PROGRAM ServoTronix
VAR_INPUT
	bExecute : REFERENCE TO BOOL;
END_VAR
VAR
	servo : AXIS_REF;
	
	mcPower : MC_Power;
	mcMoveVelocity : MC_MoveVelocity;
	mcSetPosition : MC_SetPosition;
	mcStop : MC_Stop;
	
	mcReset : MC_Reset;
	preset : BOOL;
	
	bReset : BOOL;
	positionSet : BOOL;
	
	randomPos : INT;
	
	homeLimit AT %I* : BOOL;
	home AT %I* : BOOL;
	travelLimit AT %I* : BOOL;
	
	step : (IDLE, HOME_BACK, HOME_FINAL, STOP, SET, FORWARD, REDO_HOME);
END_VAR

(*
IF NOT preset THEN
	preset := TRUE;
	bReset := TRUE;
END_IF
*)

blocks();
sequence();
IF randomPos <> 0 THEN
	mcSetPosition.Position := randomPos;
	mcSetPosition.Execute := TRUE;
	
	IF mcSetPosition.Done THEN
		mcSetPosition.Execute := FALSE;
		randomPos := 0;
	END_IF
END_IF

METHOD blocks : BOOL
mcReset(
	Axis:= servo, 
	Execute:= bReset, 
	Done=> , 
	Busy=> , 
	Error=> , 
	ErrorID=> );
	
IF bReset THEN
	bReset := FALSE;
END_IF

mcPower(
	Axis:= servo, 
	Enable:= TRUE, 
	Enable_Positive:= TRUE, 
	Enable_Negative:= TRUE, 
	Override:= 100, 
	BufferMode:= , 
	Options:= , 
	Status=> , 
	Busy=> , 
	Active=> , 
	Error=> , 
	ErrorID=> );
	
mcMoveVelocity(
	Axis:= servo, 
	Execute:= , 
	Velocity:= 75, 
	Acceleration:= , 
	Deceleration:= , 
	Jerk:= , 
	Direction:= , // MC_Positive_Direction, MC_Negative_Direction
	BufferMode:= , 
	Options:= , 
	InVelocity=> , 
	Busy=> , 
	Active=> , 
	CommandAborted=> , 
	Error=> , 
	ErrorID=> );
	
mcStop(
	Axis:= servo, 
	Execute:= , 
	Deceleration:= , 
	Jerk:= , 
	Options:= , 
	Done=> , 
	Busy=> , 
	Active=> , 
	CommandAborted=> , 
	Error=> , 
	ErrorID=> );
	
mcSetPosition(
	Axis:= servo, 
	Execute:= , 
	Position:= , 
	Mode:= , 
	Options:= , 
	Done=> , 
	Busy=> , 
	Error=> , 
	ErrorID=> );
END_METHOD

METHOD sequence : BOOL
CASE step OF
	IDLE:
		mcStop.Execute := TRUE;
		IF bExecute THEN
			bExecute := FALSE;
			mcStop.Execute := FALSE;
			
			step := HOME_BACK;
		END_IF
		
	HOME_BACK:
		mcMoveVelocity.Direction := MC_Positive_Direction;
		mcMoveVelocity.Execute := TRUE;
		
		IF NOT home THEN //if reached home
			mcMoveVelocity.Execute := FALSE;
			step := STOP;
			
		ELSIF NOT homeLimit THEN //if reached near homing limit
			mcMoveVelocity.Execute := FALSE;
			step := FORWARD;
		END_IF
		
	HOME_FINAL:
		mcMoveVelocity.Direction := MC_Negative_Direction;
		mcMoveVelocity.Execute := TRUE;
		
		IF NOT home THEN
			mcMoveVelocity.Execute := FALSE;
			step := STOP;
		END_IF
	
	STOP:
		mcStop.Execute := TRUE;
		IF mcStop.Done THEN
			mcStop.Execute := FALSE;
			step := SET;
		END_IF
		
	SET:
		mcSetPosition.Position := 0;
		mcSetPosition.Execute := TRUE;
		
		IF mcSetPosition.Done THEN
			mcSetPosition.Execute := FALSE;
			step := FORWARD;
		END_IF
	
	FORWARD:
		mcMoveVelocity.Direction := MC_Negative_Direction;
		mcMoveVelocity.Execute := TRUE;
		
		IF NOT travelLimit THEN
			
			mcMoveVelocity.Execute := FALSE;
			step := IDLE;
		END_IF
		
	REDO_HOME:
		mcMoveVelocity.Direction := MC_Negative_Direction;
		mcMoveVelocity.Execute := TRUE;
		
		IF NOT travelLimit THEN
			
			mcMoveVelocity.Execute := FALSE;
			step := HOME_BACK;
		END_IF
END_CASE
END_METHOD

END_PROGRAM

(* stored: Version 1.1.0.1, ProductVersion 3.1.4024.11
   POU ServoTronix: Id {f368819c-beba-4a2b-b26f-e222203be05a}, SpecialFunc None
   Method blocks: Id {269f953f-7162-46cc-9e48-4fb8b3aafd67}
   Method sequence: Id {86f4d543-2035-4823-a7fa-3e2e5dcf29d2} *)
